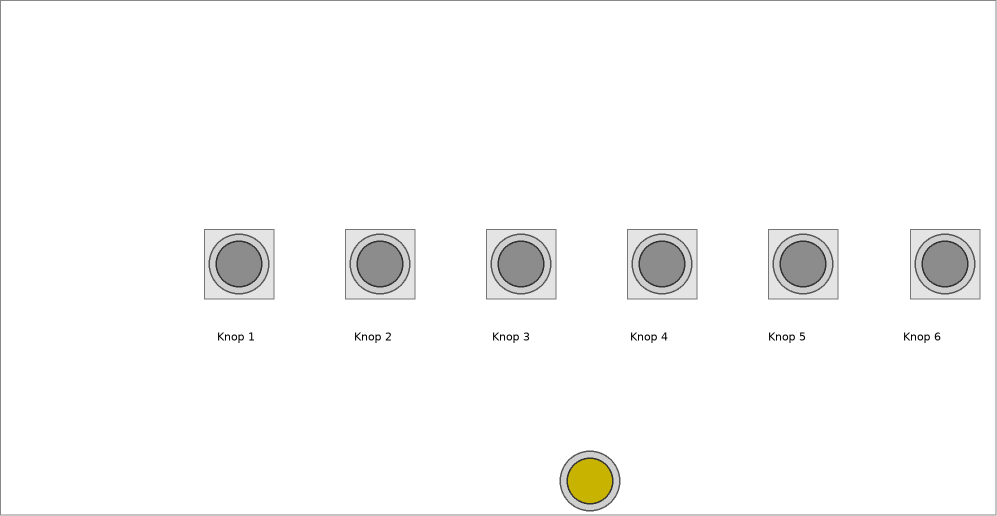
VISUALIZATION Visu  // 997x516
    PushSwitch (486,229 70x70), variable: MAIN.bKnop3, behaviour: TAP, style: Switch-PushSwitch-Gray
    PushSwitch (204,229 70x70), variable: MAIN.bKnop1, behaviour: TAP, style: Switch-PushSwitch-Gray
    PushSwitch (345,229 70x70), variable: MAIN.bKnop2, behaviour: TAP, style: Switch-PushSwitch-Gray
    PushSwitch (627,229 70x70), variable: MAIN.bKnop4, behaviour: TAP, style: Switch-PushSwitch-Gray
    PushSwitch (768,229 70x70), variable: MAIN.bKnop5, behaviour: TAP, style: Switch-PushSwitch-Gray
    PushSwitch (910,229 70x70), variable: MAIN.bKnop6, behaviour: TAP, style: Switch-PushSwitch-Gray
    Label (161,322 150x30), "Knop 1"
    Label (298,322 150x30), "Knop 2"
    Label (436,322 150x30), "Knop 3"
    Label (574,322 150x30), "Knop 4"
    Label (712,322 150x30), "Knop 5"
    Label (847,322 150x30), "Knop 6"
    Lamp1 (555,446 70x70), variable: MAIN.bLamp, style: Lamp-Lamp1-Yellow
END_VISUALIZATION

(* stored: Version 1.1.0.1, ProductVersion 3.1.4024.12
   Visu Visu: Id {8ecd5a1c-b9bd-47f1-8125-758b4fa3b6e3} *)
